{attribute 'qualified_only'}
{attribute 'strict'}
TYPE CONTROL_MODE :
(
	Off,				(*0*)
	Manual,				(*1*)
	Auto				(*2*)
);
END_TYPE

(* stored: Version 1.1.0.1
   DUT CONTROL_MODE: Id {e18a2ade-54c8-4901-a091-8c9756ab9624} *)
